FUNCTION_BLOCK AdsLogger
VAR
    Enabled : REFERENCE TO  BOOL;
END_VAR

//FB_Init is always available implicitly and it is used primarily for initialization.
//The return value is not evaluated. For a specific influence, you can also declare the
//methods explicitly and provide additional code there with the standard initialization
//code. You can evaluate the return value.
METHOD FB_Init: BOOL
VAR_INPUT
    bInitRetains: BOOL; // TRUE: the retain variables are initialized (reset warm / reset cold)
    bInCopyCode: BOOL;  // TRUE: the instance will be copied to the copy code afterward (online change) 
    Enabled : REFERENCE TO BOOL;  
END_VAR
THIS^.Enabled Ref= Enabled;
END_METHOD

METHOD LogMessage
VAR_INPUT
	Message : STRING;
END_VAR
IF THIS^.Enabled THEN
	ADSLOGSTR(ADSLOG_MSGTYPE_HINT, Message, '');
END_IF
END_METHOD

END_FUNCTION_BLOCK

(* stored: Version 1.1.0.1
   POU AdsLogger: Id {d9621f8c-9eee-45dc-90fc-0a0b1213b410}, SpecialFunc None
   Method FB_Init: Id {9b642cf8-f5ee-4a0e-955e-2a3d96f6407f}
   Method LogMessage: Id {4479acd5-067f-4d08-8bcc-fde481c11dae} *)
